FUNCTION_BLOCK OnQueueDisposedHandler EXTENDS OnQueueEventHandler

METHOD PUBLIC HandleEvent
VAR_INPUT
	Event : I_Event;
END_VAR
VAR
	queueDisposedEvent : I_QueueDisposedEvent;
END_VAR
IF __QUERYINTERFACE(Event, queueDisposedEvent) THEN
	_eventReceived := TRUE;
	fromExpected := queueDisposedEvent.TargetQueue = expectedOriginator;
END_IF
END_METHOD

END_FUNCTION_BLOCK

(* stored: Version 1.1.0.1, ProductVersion 3.1.4024.12
   POU OnQueueDisposedHandler: Id {e5ea04d5-a965-4243-b9d1-9d875c114f69}, SpecialFunc None
   Method HandleEvent: Id {502fd45b-98e3-45b4-a74b-901bd4410714} *)
